Staubli VAL3: test.dtx

mdesc mNomSpeed
mdesc mVelApprox = {accel=25, vel=50, decel=25, blend=off}
num nHPieza = 12
num nLMesa = 400
num nLPieza = 69
num nWMesa = 300
num nWPieza = 23
tool tVentosa = {z=22, fatherId=flange[0], ioLink=valve1, ioOpen=0.5, ioClose=0.5}
pointRx pCentro = {fatherId=world[0]}
pointRx pPieza = {fatherId=world[0]}
num nPlantas
num nNivel
num nFila
pointRx pObjetivo = {fatherId=world[0]}
num nX
num nY
num nZ
bool bStartPiramide
bool bTermina
jointRx jHome
bool bFin
num nTecla
string sMensaje
bool bPiezaPreparada
num nCont
num nPlantasListas
pointRx pEspera = {fatherId=world[0]}
